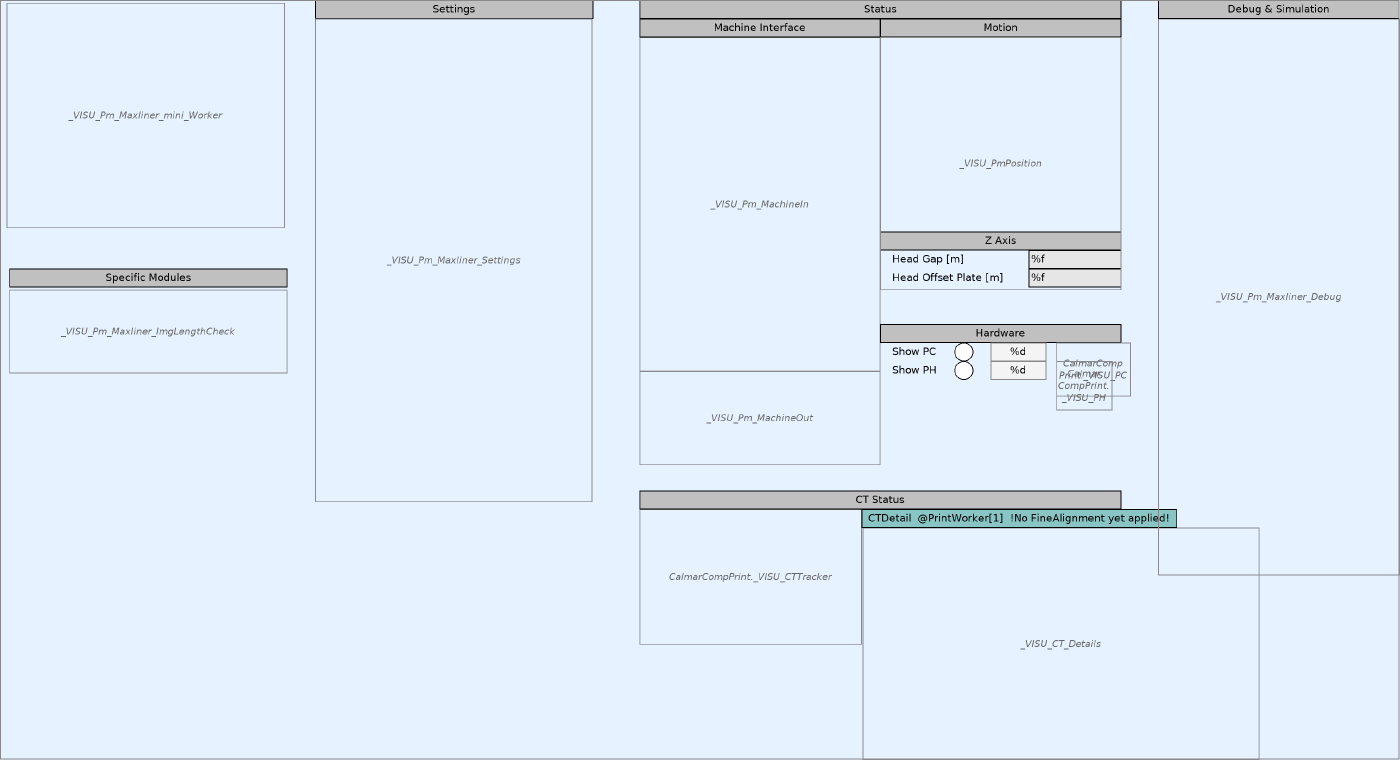
VISUALIZATION _VISU_Pm_Maxliner  // 1511x821
VAR_IN_OUT
  mInst : FB_PrintModule_Maxliner;
END_VAR
    Frame (10,313 300x90)
        shows _VISU_Pm_Maxliner_ImgLengthCheck(mInst := mInst)
    Frame (690,550 240x146)
        shows CalmarCompPrint._VISU_CTTracker(mInst := mInst.fbCTTracker)
    Frame (931,570 428x251)
        shows _VISU_CT_Details(mInst := mInst.fbWorkerPrint[1])
    Rectangle (930,550 340x20), "CTDetail @PrintWorker[1] !No FineAlignment yet applied!"
    Rectangle (690,530 520x20), "CT Status"
    Frame (690,401 260x101)
        shows _VISU_Pm_MachineOut(ref := mInst._pModuleMachineFeedback^)
    Frame (690,40 260x361)
        shows _VISU_Pm_MachineIn(ref := mInst._pModuleMachineState^)
    Rectangle (690,20 260x20), "Machine Interface"
    Rectangle (950,20 260x20), "Motion"
    Frame (7,3 300x243)
        shows _VISU_Pm_Maxliner_mini_Worker(mInst := mInst)
    Rectangle (950,350 260x20), "Hardware"
    Frame (1250,20 261x601), invisible if: NOT mInst.fbView.bShowDebugAndSim
        shows _VISU_Pm_Maxliner_Debug(mInst := mInst)
    Rectangle (340,0 300x20), "Settings"
    Rectangle (690,0 520x20), "Status"
    Rectangle (1250,0 260x20), "Debug & Simulation"
        toggle mInst.fbView.bShowDebugAndSim
    Rectangle (950,250 260x20), "Z Axis"
    Rectangle (960,270 140x20), "Head Gap [m]"
    Rectangle (1110,270 100x20), "%f", text variable: mInst._pModuleMachineFeedback^.fHeadGap
    Rectangle (960,290 140x20), "Head Offset Plate [m]"
    Rectangle (1110,290 100x20), "%f", text variable: mInst.fC_HeadOffsetPlate
    Frame (1140,370 80x58), invisible if: NOT mInst.fbView.bShowPcDetail
        shows CalmarCompPrint._VISU_PC(mInst := mInst._pPc[mInst.fbView.nSelPcDetail]^)
    Rectangle (960,390 110x20), "Show PH"
    Rectangle (960,370 110x20), "Show PC"
    Ellipse (1030,390 20x20)
        toggle mInst.fbView.bShowPhDetail
    Ellipse (1030,370 20x20)
        toggle mInst.fbView.bShowPcDetail
    Frame (1140,390 60x53), invisible if: NOT mInst.fbView.bShowPhDetail
        shows CalmarCompPrint._VISU_PH(mInst := mInst._pPh[mInst.fbView.nSelPhDetail]^)
    Scrollbar (1069,390 60x20), "%d", text variable: mInst.fbView.nSelPhDetail, invisible if: NOT mInst.fbView.bShowPhDetail
        p2245068023: mInst._nPh
        p1057716461: mInst.fbView.nSelPhDetail
    Scrollbar (1069,370 60x20), "%d", text variable: mInst.fbView.nSelPcDetail, invisible if: NOT mInst.fbView.bShowPcDetail
        p2245068023: mInst._nPc
        p1057716461: mInst.fbView.nSelPcDetail
    Rectangle (10,290 300x20), "Specific Modules"
    Frame (340,20 299x522)
        shows _VISU_Pm_Maxliner_Settings(mInst := mInst)
        p4053072137: mInst
    Frame (950,40 260x273)
        shows _VISU_PmPosition(mInst := mInst)
END_VISUALIZATION

(* stored: Version 1.1.0.1, ProductVersion 3.1.4024.11
   Visu _VISU_Pm_Maxliner: Id {620df0d7-178d-4078-9f61-c44feea74e37} *)
